(* PLC project Unnamed, Unknown Unnamed 1 *)
(* stored: creationDateTime 2025-06-21T18:09:13, modificationDateTime 2025-06-21T18:51:40 *)

PROGRAM timer_pou
  VAR
    input1 AT %IX100.0 : BOOL;
    input2 AT %IX100.1 : BOOL;
    output1 AT %QX100.0 : BOOL;
    output2 AT %QX100.1 : BOOL;
  END_VAR
  VAR
    TON0 : TON;
    TOF0 : TOF;
  END_VAR

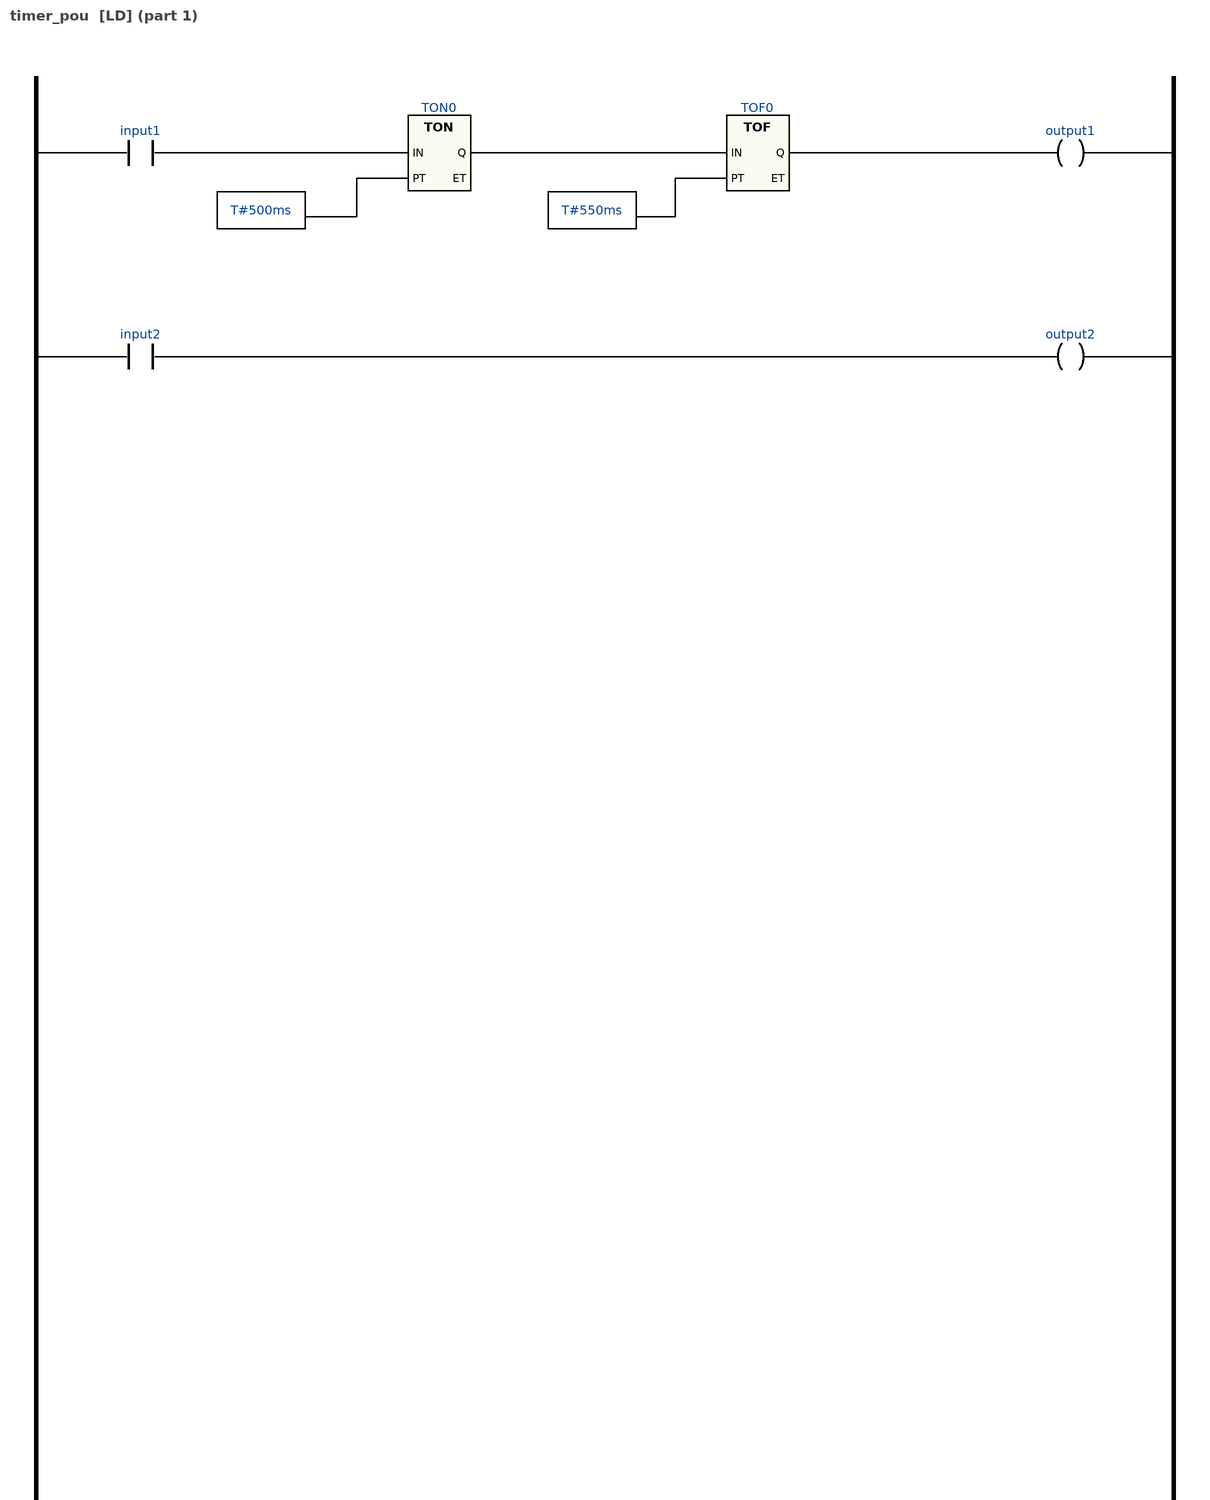
(* LD diagram, written out as Structured Text *)
TON0(IN := input1, PT := T#500ms);
TOF0(IN := TON0.Q, PT := T#550ms);
output1 := TOF0.Q;
output2 := input2;
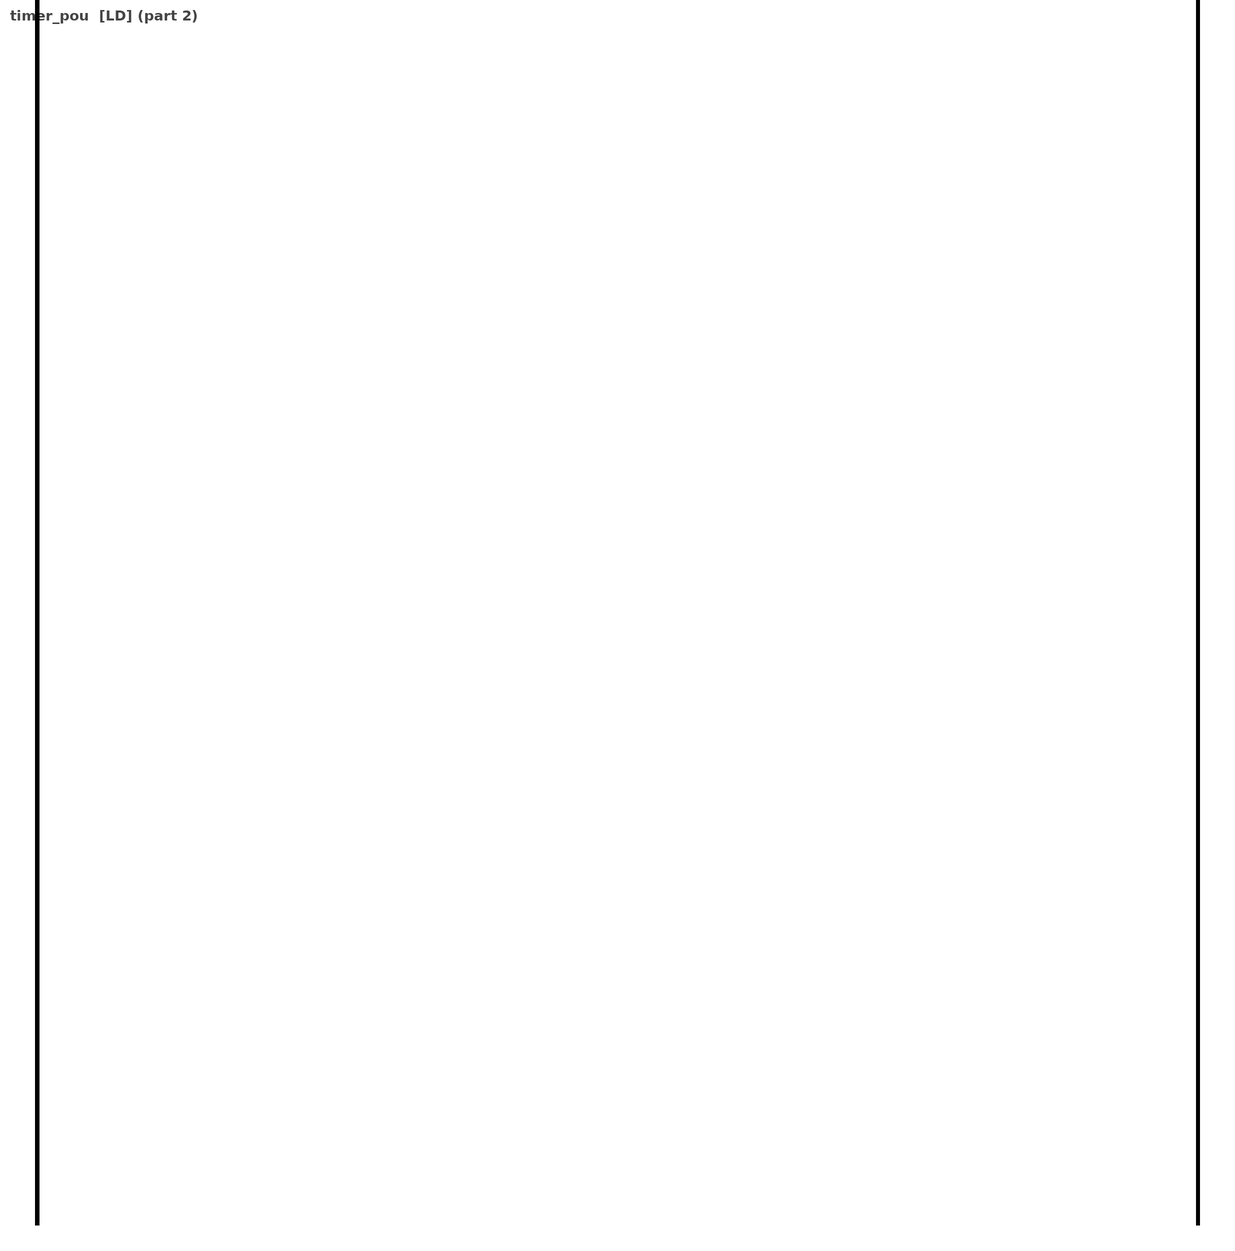
END_PROGRAM

CONFIGURATION Config0
  RESOURCE Res0 ON PLC
    TASK task0(INTERVAL := T#20ms, PRIORITY := 0);
    PROGRAM instance0 WITH task0 : timer_pou;
  END_RESOURCE
END_CONFIGURATION
